REGION Network 2 (SCL): Data to HMI
   "HMI_BUTTON_START_KPPU" := "MB_BUTTON_START_KPPU";
   "HMI_BUTTON_STOP_KPPU" := "MB_BUTTON_STOP_KPPU";
   "HMI_MODE_auto" := "Global".MODE_auto;
   "HMI_MODE_manual" := "Global".MODE_manual;
   "HMI_MODE_blocked" := "Global".MODE_blocked;
   "HMI_MODE_standby" := "Global".MODE_standby;
   "HMI_MODE_standby_pressure_high" := "Global".MODE_standby_pressure_high;
   "HMI_BUTTON_Global_Stop" := "Global".BUTTON_Global_Stop;
   "HMI_Global_Stop" := "Global".Global_Stop;
   "HMI_BUTTON_Sound_Off" := "Global".BUTTON_Sound_Off;
   "HMI_BUTTON_Led_Test" := "Global".BUTTON_Led_Test;
   "HMI_STATE_380_main" := "Global".STATE_380_main;
   "HMI_STATE_380_backup" := "Global".STATE_380_backup;
   "HMI_STATE_220_inner" := "Global".STATE_220_inner;
   "HMI_STATE_220_outer" := "Global".STATE_220_outer;
   "HMI_STATE_door_opened" := "Global".STATE_door_opened;
   "HMI_ERROR_underwater" := "Global".ERROR_underwater;
   "HMI_ERROR_no_water" := "Global".ERROR_no_water;
   "HMI_ERROR_no_water_fire" := "Global".ERROR_no_water_fire;
   "HMI_ERROR_inlet_pressure_low" := "Global".ERROR_inlet_pressure_low;
   "HMI_ERROR_global" := "Global".ERROR_global;
   "HMI_ERROR_Main_Ball_Valves" := "Global".ERROR_Main_Ball_Valves;
   "HMI_ERROR_BALL_VALVE_ANY" := "Global".ERROR_BALL_VALVE_ANY;
   "HMI_ERROR_any" := "Global".ERROR_any;
   "HMI_SIGNAL_fire" := "Global".SIGNAL_fire;
   "HMI_SIGNAL_fire_by_pressure" := "Global".SIGNAL_fire_by_pressure;
   "HMI_ERROR_high_pressure_redundancy" := "Global".ERROR_high_pressure_redundancy;
   "HMI_ERROR_low_pressure_redundancy" := "Global".ERROR_low_pressure_redundancy;
   "HMI_SIGNAL_first_pump_has_started" := "Global".SIGNAL_first_pump_has_started;
   "HMI_Start_standby_pump" := "Global".Start_standby_pump;
   "HMI_Secret_condition" := "Global".Secret_condition;
   "HMI_ERROR_Battery_low" := "Global".ERROR_Battery_low;
   "HMI_ERROR_connection_lost" := "Global".ERROR_connection_lost;
   "HMI_ERROR_connection_lost_TOF" := "Global".ERROR_connection_lost_TOF;
   "HMI_ERROR_connection_lost_TON" := "Global".ERROR_connection_lost_TON;
   "HMI_SENSOR_low_pressure_PIS1.1_error" := "Global"."SENSOR_low_pressure_PIS1.1_error";
   "HMI_SENSOR_low_pressure_PIS1.2_error" := "Global"."SENSOR_low_pressure_PIS1.2_error";
   "HMI_SENSOR_high_pressure_PIS2.1_error" := "Global"."SENSOR_high_pressure_PIS2.1_error";
   "HMI_SENSOR_high_pressure_PIS2.2_error" := "Global"."SENSOR_high_pressure_PIS2.2_error";
   "HMI_IN_valve_gate__ERROR_B1" := "Low_pressure_valves"."IN_valve_gate__ERROR_B"[1];
   "HMI_IN_valve_gate__ERROR_B2" := "Low_pressure_valves"."IN_valve_gate__ERROR_B"[2];
   "HMI_IN_valve_gate__ERROR_B3" := "Low_pressure_valves"."IN_valve_gate__ERROR_B"[3];
   "HMI_IN_valve_gate__ERROR_B4" := "Low_pressure_valves"."IN_valve_gate__ERROR_B"[4];
   "HMI_IN_valve_gate__ERROR_B5" := "Low_pressure_valves"."IN_valve_gate__ERROR_B"[5];
   "HMI_IN_valve_gate__ERROR_B6" := "Low_pressure_valves"."IN_valve_gate__ERROR_B"[6];
   "HMI_IN_valve_gate__ERROR_B7" := "Low_pressure_valves"."IN_valve_gate__ERROR_B"[7];
   "HMI_IN_valve_gate__ERROR_B8" := "Low_pressure_valves"."IN_valve_gate__ERROR_B"[8];
   "HMI_IN_valve_gate__ERROR_B9" := "Low_pressure_valves"."IN_valve_gate__ERROR_B"[9];
   "HMI_ERROR_IN_VALVE_ANY" := "Low_pressure_valves".ERROR_IN_VALVE_ANY;
   "HMI_SENSOR_flow_UUS1" := "Section_valves_data".SENSOR_flow_UUS[1];
   "HMI_SENSOR_flow_UUS2" := "Section_valves_data".SENSOR_flow_UUS[2];
   "HMI_SENSOR_flow_UUS3" := "Section_valves_data".SENSOR_flow_UUS[3];
   "HMI_SENSOR_flow_UUS4" := "Section_valves_data".SENSOR_flow_UUS[4];
   "HMI_ERROR_UUS1" := "Section_valves_data".ERROR_UUS[1];
   "HMI_ERROR_UUS2" := "Section_valves_data".ERROR_UUS[2];
   "HMI_ERROR_UUS3" := "Section_valves_data".ERROR_UUS[3];
   "HMI_ERROR_UUS4" := "Section_valves_data".ERROR_UUS[4];
   "HMI_ERROR_UUS_ANY" := "Section_valves_data".ERROR_UUS_ANY;
   "HMI_ERROR_UUS_ALL" := "Section_valves_data".ERROR_UUS_ALL;
   "HMI_State_switch_pump1" := "Pumps_data".State_switch_pump[1];
   "HMI_State_switch_pump2" := "Pumps_data".State_switch_pump[2];
   "HMI_State_switch_pump3" := "Pumps_data".State_switch_pump[3];
   "HMI_State_switch_pump4" := "Pumps_data".State_switch_pump[4];
   "HMI_State_switch_pump5" := "Pumps_data".State_switch_pump[5];
   "HMI_Error_pump1" := "Pumps_data".Error_pump[1];
   "HMI_Error_pump2" := "Pumps_data".Error_pump[2];
   "HMI_Error_pump3" := "Pumps_data".Error_pump[3];
   "HMI_Error_pump4" := "Pumps_data".Error_pump[4];
   "HMI_Error_pump5" := "Pumps_data".Error_pump[5];
   "HMI_State_starter_pump1" := "Pumps_data".State_starter_pump[1];
   "HMI_State_starter_pump2" := "Pumps_data".State_starter_pump[2];
   "HMI_State_starter_pump3" := "Pumps_data".State_starter_pump[3];
   "HMI_State_starter_pump4" := "Pumps_data".State_starter_pump[4];
   "HMI_State_starter_pump5" := "Pumps_data".State_starter_pump[5];
   "HMI_State_work_pump1" := "Pumps_data".State_work_pump[1];
   "HMI_State_work_pump2" := "Pumps_data".State_work_pump[2];
   "HMI_State_work_pump3" := "Pumps_data".State_work_pump[3];
   "HMI_State_work_pump4" := "Pumps_data".State_work_pump[4];
   "HMI_State_work_pump5" := "Pumps_data".State_work_pump[5];
   "HMI_Pump_pressure_sensor_error1" := "Pumps_data".Pump_pressure_sensor_error[1];
   "HMI_Pump_pressure_sensor_error2" := "Pumps_data".Pump_pressure_sensor_error[2];
   "HMI_Pump_pressure_sensor_error3" := "Pumps_data".Pump_pressure_sensor_error[3];
   "HMI_Pump_pressure_sensor_error4" := "Pumps_data".Pump_pressure_sensor_error[4];
   "HMI_Pump_pressure_sensor_error5" := "Pumps_data".Pump_pressure_sensor_error[5];
   "HMI_State_switch_standby_pump" := "Pumps_data".State_switch_standby_pump;
   "HMI_Error_any_pump" := "Pumps_data".Error_any_pump;
   "HMI_Error_standby_pump" := "Pumps_data".Error_standby_pump;
   "HMI_State_starter_standby_pump" := "Pumps_data".State_starter_standby_pump;
   "HMI_State_work_standby_pump" := "Pumps_data".State_work_standby_pump;
   "HMI_State_work_any_pump" := "Pumps_data".State_work_any_pump;
   "HMI_ERROR_PUMPS_ANY" := "Pumps_data".ERROR_PUMPS_ANY;
   "HMI_ERROR_PUMPS_ALL" := "Pumps_data".ERROR_PUMPS_ALL;
   "HMI_Low_pressure_valve_B1_open_OFF" := "SOVA_Modbus_Input".MB_Line[1, 1, 0];
   "HMI_Low_pressure_valve_B1_open_NO_signal" := "SOVA_Modbus_Input".MB_Line[1, 1, 1];
   "HMI_Low_pressure_valve_B1_open_short" := "SOVA_Modbus_Input".MB_Line[1, 1, 4];
   "HMI_Low_pressure_valve_B1_open_brake" := "SOVA_Modbus_Input".MB_Line[1, 1, 5];
   "HMI_Low_pressure_valve_B1_open_Signal" := "SOVA_Modbus_Input".MB_Line[1, 1, 6];
   "HMI_Low_pressure_valve_B1_close_OFF" := "SOVA_Modbus_Input".MB_Line[1, 2, 0];
   "HMI_Low_pressure_valve_B1_close_NO_signal" := "SOVA_Modbus_Input".MB_Line[1, 2, 1];
   "HMI_Low_pressure_valve_B1_close_short" := "SOVA_Modbus_Input".MB_Line[1, 2, 4];
   "HMI_Low_pressure_valve_B1_close_brake" := "SOVA_Modbus_Input".MB_Line[1, 2, 5];
   "HMI_Low_pressure_valve_B1_close_Signal" := "SOVA_Modbus_Input".MB_Line[1, 2, 6];
   "HMI_Low_pressure_valve_B2_open_OFF" := "SOVA_Modbus_Input".MB_Line[1, 3, 0];
   "HMI_Low_pressure_valve_B2_open_NO_signal" := "SOVA_Modbus_Input".MB_Line[1, 3, 1];
   "HMI_Low_pressure_valve_B2_open_short" := "SOVA_Modbus_Input".MB_Line[1, 3, 4];
   "HMI_Low_pressure_valve_B2_open_brake" := "SOVA_Modbus_Input".MB_Line[1, 3, 5];
   "HMI_Low_pressure_valve_B2_open_Signal" := "SOVA_Modbus_Input".MB_Line[1, 3, 6];
   "HMI_Low_pressure_valve_B2_close_OFF" := "SOVA_Modbus_Input".MB_Line[1, 4, 0];
   "HMI_Low_pressure_valve_B2_close_NO_signal" := "SOVA_Modbus_Input".MB_Line[1, 4, 1];
   "HMI_Low_pressure_valve_B2_close_short" := "SOVA_Modbus_Input".MB_Line[1, 4, 4];
   "HMI_Low_pressure_valve_B2_close_brake" := "SOVA_Modbus_Input".MB_Line[1, 4, 5];
   "HMI_Low_pressure_valve_B2_close_Signal" := "SOVA_Modbus_Input".MB_Line[1, 4, 6];
   "HMI_Low_pressure_valve_B3_open_OFF" := "SOVA_Modbus_Input".MB_Line[1, 5, 0];
   "HMI_Low_pressure_valve_B3_open_NO_signal" := "SOVA_Modbus_Input".MB_Line[1, 5, 1];
   "HMI_Low_pressure_valve_B3_open_short" := "SOVA_Modbus_Input".MB_Line[1, 5, 4];
   "HMI_Low_pressure_valve_B3_open_brake" := "SOVA_Modbus_Input".MB_Line[1, 5, 5];
   "HMI_Low_pressure_valve_B3_open_Signal" := "SOVA_Modbus_Input".MB_Line[1, 5, 6];
   "HMI_Low_pressure_valve_B3_close_OFF" := "SOVA_Modbus_Input".MB_Line[1, 6, 0];
   "HMI_Low_pressure_valve_B3_close_NO_signal" := "SOVA_Modbus_Input".MB_Line[1, 6, 1];
   "HMI_Low_pressure_valve_B3_close_short" := "SOVA_Modbus_Input".MB_Line[1, 6, 4];
   "HMI_Low_pressure_valve_B3_close_brake" := "SOVA_Modbus_Input".MB_Line[1, 6, 5];
   "HMI_Low_pressure_valve_B3_close_Signal" := "SOVA_Modbus_Input".MB_Line[1, 6, 6];
   "HMI_Low_pressure_valve_B4_open_OFF" := "SOVA_Modbus_Input".MB_Line[1, 7, 0];
   "HMI_Low_pressure_valve_B4_open_NO_signal" := "SOVA_Modbus_Input".MB_Line[1, 7, 1];
   "HMI_Low_pressure_valve_B4_open_short" := "SOVA_Modbus_Input".MB_Line[1, 7, 4];
   "HMI_Low_pressure_valve_B4_open_brake" := "SOVA_Modbus_Input".MB_Line[1, 7, 5];
   "HMI_Low_pressure_valve_B4_open_Signal" := "SOVA_Modbus_Input".MB_Line[1, 7, 6];
   "HMI_Low_pressure_valve_B4_close_OFF" := "SOVA_Modbus_Input".MB_Line[1, 8, 0];
   "HMI_Low_pressure_valve_B4_close_NO_signal" := "SOVA_Modbus_Input".MB_Line[1, 8, 1];
   "HMI_Low_pressure_valve_B4_close_short" := "SOVA_Modbus_Input".MB_Line[1, 8, 4];
   "HMI_Low_pressure_valve_B4_close_brake" := "SOVA_Modbus_Input".MB_Line[1, 8, 5];
   "HMI_Low_pressure_valve_B4_close_Signal" := "SOVA_Modbus_Input".MB_Line[1, 8, 6];
   "HMI_Low_pressure_valve_B5_open_OFF" := "SOVA_Modbus_Input".MB_Line[1, 9, 0];
   "HMI_Low_pressure_valve_B5_open_NO_signal" := "SOVA_Modbus_Input".MB_Line[1, 9, 1];
   "HMI_Low_pressure_valve_B5_open_short" := "SOVA_Modbus_Input".MB_Line[1, 9, 4];
   "HMI_Low_pressure_valve_B5_open_brake" := "SOVA_Modbus_Input".MB_Line[1, 9, 5];
   "HMI_Low_pressure_valve_B5_open_Signal" := "SOVA_Modbus_Input".MB_Line[1, 9, 6];
   "HMI_Low_pressure_valve_B5_close_OFF" := "SOVA_Modbus_Input".MB_Line[1, 10, 0];
   "HMI_Low_pressure_valve_B5_close_NO_signal" := "SOVA_Modbus_Input".MB_Line[1, 10, 1];
   "HMI_Low_pressure_valve_B5_close_short" := "SOVA_Modbus_Input".MB_Line[1, 10, 4];
   "HMI_Low_pressure_valve_B5_close_brake" := "SOVA_Modbus_Input".MB_Line[1, 10, 5];
   "HMI_Low_pressure_valve_B5_close_Signal" := "SOVA_Modbus_Input".MB_Line[1, 10, 6];
   "HMI_Low_pressure_valve_B6_open_OFF" := "SOVA_Modbus_Input".MB_Line[1, 11, 0];
   "HMI_Low_pressure_valve_B6_open_NO_signal" := "SOVA_Modbus_Input".MB_Line[1, 11, 1];
   "HMI_Low_pressure_valve_B6_open_short" := "SOVA_Modbus_Input".MB_Line[1, 11, 4];
   "HMI_Low_pressure_valve_B6_open_brake" := "SOVA_Modbus_Input".MB_Line[1, 11, 5];
   "HMI_Low_pressure_valve_B6_open_Signal" := "SOVA_Modbus_Input".MB_Line[1, 11, 6];
   "HMI_Low_pressure_valve_B6_close_OFF" := "SOVA_Modbus_Input".MB_Line[1, 12, 0];
   "HMI_Low_pressure_valve_B6_close_NO_signal" := "SOVA_Modbus_Input".MB_Line[1, 12, 1];
   "HMI_Low_pressure_valve_B6_close_short" := "SOVA_Modbus_Input".MB_Line[1, 12, 4];
   "HMI_Low_pressure_valve_B6_close_brake" := "SOVA_Modbus_Input".MB_Line[1, 12, 5];
   "HMI_Low_pressure_valve_B6_close_Signal" := "SOVA_Modbus_Input".MB_Line[1, 12, 6];
   "HMI_Low_pressure_valve_B7_open_OFF" := "SOVA_Modbus_Input".MB_Line[2, 1, 0];
   "HMI_Low_pressure_valve_B7_open_NO_signal" := "SOVA_Modbus_Input".MB_Line[2, 1, 1];
   "HMI_Low_pressure_valve_B7_open_short" := "SOVA_Modbus_Input".MB_Line[2, 1, 4];
   "HMI_Low_pressure_valve_B7_open_brake" := "SOVA_Modbus_Input".MB_Line[2, 1, 5];
   "HMI_Low_pressure_valve_B7_open_Signal" := "SOVA_Modbus_Input".MB_Line[2, 1, 6];
   "HMI_Low_pressure_valve_B7_close_OFF" := "SOVA_Modbus_Input".MB_Line[2, 2, 0];
   "HMI_Low_pressure_valve_B7_close_NO_signal" := "SOVA_Modbus_Input".MB_Line[2, 2, 1];
   "HMI_Low_pressure_valve_B7_close_short" := "SOVA_Modbus_Input".MB_Line[2, 2, 4];
   "HMI_Low_pressure_valve_B7_close_brake" := "SOVA_Modbus_Input".MB_Line[2, 2, 5];
   "HMI_Low_pressure_valve_B7_close_Signal" := "SOVA_Modbus_Input".MB_Line[2, 2, 6];
   "HMI_Low_pressure_valve_B8_open_OFF" := "SOVA_Modbus_Input".MB_Line[2, 3, 0];
   "HMI_Low_pressure_valve_B8_open_NO_signal" := "SOVA_Modbus_Input".MB_Line[2, 3, 1];
   "HMI_Low_pressure_valve_B8_open_short" := "SOVA_Modbus_Input".MB_Line[2, 3, 4];
   "HMI_Low_pressure_valve_B8_open_brake" := "SOVA_Modbus_Input".MB_Line[2, 3, 5];
   "HMI_Low_pressure_valve_B8_open_Signal" := "SOVA_Modbus_Input".MB_Line[2, 3, 6];
   "HMI_Low_pressure_valve_B8_close_OFF" := "SOVA_Modbus_Input".MB_Line[2, 4, 0];
   "HMI_Low_pressure_valve_B8_close_NO_signal" := "SOVA_Modbus_Input".MB_Line[2, 4, 1];
   "HMI_Low_pressure_valve_B8_close_short" := "SOVA_Modbus_Input".MB_Line[2, 4, 4];
   "HMI_Low_pressure_valve_B8_close_brake" := "SOVA_Modbus_Input".MB_Line[2, 4, 5];
   "HMI_Low_pressure_valve_B8_close_Signal" := "SOVA_Modbus_Input".MB_Line[2, 4, 6];
   "HMI_Low_pressure_valve_B9_open_OFF" := "SOVA_Modbus_Input".MB_Line[2, 5, 0];
   "HMI_Low_pressure_valve_B9_open_NO_signal" := "SOVA_Modbus_Input".MB_Line[2, 5, 1];
   "HMI_Low_pressure_valve_B9_open_short" := "SOVA_Modbus_Input".MB_Line[2, 5, 4];
   "HMI_Low_pressure_valve_B9_open_brake" := "SOVA_Modbus_Input".MB_Line[2, 5, 5];
   "HMI_Low_pressure_valve_B9_open_Signal" := "SOVA_Modbus_Input".MB_Line[2, 5, 6];
   "HMI_Low_pressure_valve_B9_close_OFF" := "SOVA_Modbus_Input".MB_Line[2, 6, 0];
   "HMI_Low_pressure_valve_B9_close_NO_signal" := "SOVA_Modbus_Input".MB_Line[2, 6, 1];
   "HMI_Low_pressure_valve_B9_close_short" := "SOVA_Modbus_Input".MB_Line[2, 6, 4];
   "HMI_Low_pressure_valve_B9_close_brake" := "SOVA_Modbus_Input".MB_Line[2, 6, 5];
   "HMI_Low_pressure_valve_B9_close_Signal" := "SOVA_Modbus_Input".MB_Line[2, 6, 6];
   "HMI_Ball_valve_K38.1_open_OFF" := "SOVA_Modbus_Input".MB_Line[3, 1, 0];
   "HMI_Ball_valve_K38.1_open_NO_signal" := "SOVA_Modbus_Input".MB_Line[3, 1, 1];
   "HMI_Ball_valve_K38.1_open_short" := "SOVA_Modbus_Input".MB_Line[3, 1, 4];
   "HMI_Ball_valve_K38.1_open_brake" := "SOVA_Modbus_Input".MB_Line[3, 1, 5];
   "HMI_Ball_valve_K38.1_open_Signal" := "SOVA_Modbus_Input".MB_Line[3, 1, 6];
   "HMI_Ball_valve_K38.2_open_OFF" := "SOVA_Modbus_Input".MB_Line[3, 2, 0];
   "HMI_Ball_valve_K38.2_open_NO_signal" := "SOVA_Modbus_Input".MB_Line[3, 2, 1];
   "HMI_Ball_valve_K38.2_open_short" := "SOVA_Modbus_Input".MB_Line[3, 2, 4];
   "HMI_Ball_valve_K38.2_open_brake" := "SOVA_Modbus_Input".MB_Line[3, 2, 5];
   "HMI_Ball_valve_K38.2_open_Signal" := "SOVA_Modbus_Input".MB_Line[3, 2, 6];
   "HMI_Ball_valve_K38.3_open_OFF" := "SOVA_Modbus_Input".MB_Line[3, 3, 0];
   "HMI_Ball_valve_K38.3_open_NO_signal" := "SOVA_Modbus_Input".MB_Line[3, 3, 1];
   "HMI_Ball_valve_K38.3_open_short" := "SOVA_Modbus_Input".MB_Line[3, 3, 4];
   "HMI_Ball_valve_K38.3_open_brake" := "SOVA_Modbus_Input".MB_Line[3, 3, 5];
   "HMI_Ball_valve_K38.3_open_Signal" := "SOVA_Modbus_Input".MB_Line[3, 3, 6];
   "HMI_Ball_valve_K38.4_open_OFF" := "SOVA_Modbus_Input".MB_Line[3, 4, 0];
   "HMI_Ball_valve_K38.4_open_NO_signal" := "SOVA_Modbus_Input".MB_Line[3, 4, 1];
   "HMI_Ball_valve_K38.4_open_short" := "SOVA_Modbus_Input".MB_Line[3, 4, 4];
   "HMI_Ball_valve_K38.4_open_brake" := "SOVA_Modbus_Input".MB_Line[3, 4, 5];
   "HMI_Ball_valve_K38.4_open_Signal" := "SOVA_Modbus_Input".MB_Line[3, 4, 6];
   "HMI_Ball_valve_K38.5_open_OFF" := "SOVA_Modbus_Input".MB_Line[3, 5, 0];
   "HMI_Ball_valve_K38.5_open_NO_signal" := "SOVA_Modbus_Input".MB_Line[3, 5, 1];
   "HMI_Ball_valve_K38.5_open_short" := "SOVA_Modbus_Input".MB_Line[3, 5, 4];
   "HMI_Ball_valve_K38.5_open_brake" := "SOVA_Modbus_Input".MB_Line[3, 5, 5];
   "HMI_Ball_valve_K38.5_open_Signal" := "SOVA_Modbus_Input".MB_Line[3, 5, 6];
   "HMI_UUS.1_open_OFF" := "SOVA_Modbus_Input".MB_Line[3, 7, 0];
   "HMI_UUS.1_open_NO_signal" := "SOVA_Modbus_Input".MB_Line[3, 7, 1];
   "HMI_UUS.1_open_short" := "SOVA_Modbus_Input".MB_Line[3, 7, 4];
   "HMI_UUS.1_open_brake" := "SOVA_Modbus_Input".MB_Line[3, 7, 5];
   "HMI_UUS.1_open_Signal" := "SOVA_Modbus_Input".MB_Line[3, 7, 6];
   "HMI_UUS.2_open_OFF" := "SOVA_Modbus_Input".MB_Line[3, 8, 0];
   "HMI_UUS.2_open_NO_signal" := "SOVA_Modbus_Input".MB_Line[3, 8, 1];
   "HMI_UUS.2_open_short" := "SOVA_Modbus_Input".MB_Line[3, 8, 4];
   "HMI_UUS.2_open_brake" := "SOVA_Modbus_Input".MB_Line[3, 8, 5];
   "HMI_UUS.2_open_Signal" := "SOVA_Modbus_Input".MB_Line[3, 8, 6];
   "HMI_UUS.3_open_OFF" := "SOVA_Modbus_Input".MB_Line[3, 9, 0];
   "HMI_UUS.3_open_NO_signal" := "SOVA_Modbus_Input".MB_Line[3, 9, 1];
   "HMI_UUS.3_open_short" := "SOVA_Modbus_Input".MB_Line[3, 9, 4];
   "HMI_UUS.3_open_brake" := "SOVA_Modbus_Input".MB_Line[3, 9, 5];
   "HMI_UUS.3_open_Signal" := "SOVA_Modbus_Input".MB_Line[3, 9, 6];
   "HMI_UUS.4_open_OFF" := "SOVA_Modbus_Input".MB_Line[3, 10, 0];
   "HMI_UUS.4_open_NO_signal" := "SOVA_Modbus_Input".MB_Line[3, 10, 1];
   "HMI_UUS.4_open_short" := "SOVA_Modbus_Input".MB_Line[3, 10, 4];
   "HMI_UUS.4_open_brake" := "SOVA_Modbus_Input".MB_Line[3, 10, 5];
   "HMI_UUS.4_open_Signal" := "SOVA_Modbus_Input".MB_Line[3, 10, 6];
   "HMI_SENSOR_low_pressure_PIS1.1" := "Global"."SENSOR_low_pressure_PIS1.1";
   "HMI_SENSOR_low_pressure_PIS1.2" := "Global"."SENSOR_low_pressure_PIS1.2";
   "HMI_SENSOR_high_pressure_PIS2.1" := "Global"."SENSOR_high_pressure_PIS2.1";
   "HMI_SENSOR_high_pressure_PIS2.2" := "Global"."SENSOR_high_pressure_PIS2.2";
   "HMI_INDICATION_high_pressure" := "Global".INDICATION_high_pressure;
   "HMI_INDICATION_low_pressure" := "Global".INDICATION_low_pressure;
   "HMI_Pump_pressure_sensor1" := "Pumps_data".Pump_pressure_sensor[1];
   "HMI_Pump_pressure_sensor2" := "Pumps_data".Pump_pressure_sensor[2];
   "HMI_Pump_pressure_sensor3" := "Pumps_data".Pump_pressure_sensor[3];
   "HMI_Pump_pressure_sensor4" := "Pumps_data".Pump_pressure_sensor[4];
   "HMI_Pump_pressure_sensor5" := "Pumps_data".Pump_pressure_sensor[5];
END_REGION
END_ORGANIZATION_BLOCK